FUNCTION_BLOCK FB_CN_CentralMachineCooling EXTENDS FB_SystemContinous
VAR_INPUT
END_VAR
VAR_OUTPUT
END_VAR
VAR
	//default parameters
	localDefaultParameters : ST_CN_CentralMachineCoolingDefaultParameters;
	
	//pumps
	stPU100DefaultParameters : ST_PumpGrundfosMagna3DefaultParameters := (tTaskCycleTime := GlobalVariables.tTaskCycleTime_MAIN, tCtrlCycleTime := GlobalVariables.tCtrlCycleTime_MAIN);
	PU100 : FB_PumpGrundfosMagna3 := (ST_DefaultParameters := stPU100DefaultParameters);;

	//valves
	stSV100DefaultParameters : ST_DiscreteValveDefaultParameters := (nFeedback := 3);
	SV100 : FB_DiscreteValve := (ST_DefaultParameters := stSV100DefaultParameters);
	
	WMZ100: FB_MollineEHeatCounter;
	
	//internal variables
	bSetStatusOn_PU100 : BOOL;
	bSetStatusOn_SV100 : BOOL;
END_VAR

MAIN();

SV100.GetState_BI();
SV100(bSetStatusOnAutomatic := bSetStatusOn_SV100,
	bAlgorithmPermission := bAlgorithmPermission);
SV100.SetState_BO();

//pump controls return temperature
PU100.GetState_Profibus();
PU100(bSetStatusOnAutomatic := bSetStatusOn_PU100,
	bAlgorithmPermission := bAlgorithmPermission,
	fSetPointAutomatic := fSetPoint,
	nControlModeAutomatic := 1);
PU100.SetState_Profibus();

WMZ100(aHeatCounterTelegramm:=aTelegramm_WMZ100);

METHOD PROTECTED  CheckError : BOOL
VAR_INPUT
END_VAR
VAR_OUTPUT
	bError : BOOL;
END_VAR
IF (PU100.bStatusOn AND SV100.localState.nPosition = 2) OR PU100.bError THEN
	bError := TRUE;
END_IF
END_METHOD

METHOD PROTECTED  Operational : BOOL
VAR_INPUT
END_VAR
VAR_OUTPUT
	bSwitchToWorking : BOOL := FALSE;
END_VAR
bSetStatusOn_PU100 := TRUE;

IF PU100.bStatusOn THEN
	bSwitchToWorking := TRUE;
END_IF
END_METHOD

METHOD PROTECTED  RampDown : BOOL
VAR_INPUT
END_VAR
VAR_OUTPUT
	bRampDownFinished : BOOL := FALSE;
END_VAR
bSetStatusOn_PU100 := FALSE;

IF NOT PU100.bStatusOn THEN
	bSetStatusOn_SV100 := FALSE;
	IF SV100.localState.nPosition = 2 THEN
		bRampDownFinished := TRUE;
	END_IF
END_IF
END_METHOD

METHOD PROTECTED  RampUp : BOOL
VAR_INPUT
END_VAR
VAR_OUTPUT
	bRampUpFinished : BOOL := FALSE;
END_VAR
bSetStatusOn_SV100 := TRUE;

IF SV100.localState.nPosition = 3 THEN
	bRampUpFinished := TRUE;
END_IF
END_METHOD

METHOD PROTECTED   SetSetPointLimits : BOOL
VAR_INPUT
END_VAR
aSetPointLimits[1] := localDefaultParameters.aSetPointLimitsTemperature[1];
aSetPointLimits[2] := localDefaultParameters.aSetPointLimitsTemperature[2];
END_METHOD

METHOD PROTECTED  SetState : BOOL
VAR_INPUT
END_VAR
VAR_OUTPUT
END_VAR
fOperatingPoint := PU100.fTemperatureExternal;

controlState.bStatusOn := bSetStatusOn;
setPointState.aSetPointLimits := aSetPointLimits;
setPointState.fSetPoint := fSetPoint;
setPointState.fOperatingPoint := fOperatingPoint;
setPointState.sSetPointUnit := 'degreeC';
setPointState.sOperatingPointUnit := 'degreeC';
END_METHOD

METHOD PROTECTED  Working : BOOL
VAR_INPUT
END_VAR
VAR_OUTPUT
	bSwitchToOperational : BOOL := FALSE;
END_VAR
//empty method
END_METHOD

END_FUNCTION_BLOCK

(* stored: Version 1.1.0.1, ProductVersion 3.1.4024.10
   POU FB_CN_CentralMachineCooling: Id {0a11f1d0-fdb2-4a95-b568-34fd403f1a7b}, SpecialFunc None
   Method CheckError: Id {4276cf4c-f380-44a1-8219-8445a723854b}
   Method Operational: Id {d90af776-5306-44f7-8360-e5330d395bda}
   Method RampDown: Id {7afd6cbf-89bd-40f8-b6d2-a42b5171e63e}
   Method RampUp: Id {7d5405b2-d5ca-46b6-81e3-1ffe28574586}
   Method SetSetPointLimits: Id {6ce66674-d039-4ebc-9baf-9c2d93b0cf06}
   Method SetState: Id {070992e0-f9f9-47d5-b026-51312d817469}
   Method Working: Id {841d2a3c-59fc-4555-9ce9-0f784f18eb2c} *)
